{attribute 'qualified_only'}
{attribute 'strict'}
TYPE eCheckResult :
(
    None := 0,
    Passed := 10,
    Failed := 20
);
END_TYPE

(* stored: Version 1.1.0.1, ProductVersion 3.1.4024.9
   DUT eCheckResult: Id {7531f9dc-26cd-4c0e-a6f8-2481f0149d69} *)
